PROGRAM MAIN
VAR
	bIsInitialized	: BOOL;
	//Alarms 
	fbAlarm1		: FB_TcAlarm;
	fbAlarm2		: FB_TcAlarm;
	fbAlarm3		: FB_TcAlarm;
	fbAlarm4		: FB_TcAlarm;
	fbAlarm5		: FB_TcAlarm;
	bAlarm			: BOOL;
	bClearAlarm		: BOOL;
	//Warning 
	fbWarning1 		: FB_TcAlarm;
	fbWarning2 		: FB_TcAlarm;
	fbWarning3 		: FB_TcAlarm;
	fbWarning4 		: FB_TcAlarm;
	fbWarning5 		: FB_TcAlarm;
	bWarning		: BOOL;
	bClearWarning	: BOOL;
	//Info
	fbInfo1			: FB_TcMessage;
	fbInfo2			: FB_TcMessage;
	fbInfo3			: FB_TcMessage;
	fbInfo4			: FB_TcMessage;
	fbInfo5			: FB_TcMessage;	
	bInfo			: BOOL;
	//To show alarms with arguments
	fbAlarmWithArgument1 	: FB_TcAlarm;
	fbAlarmWithArgument2 	: FB_TcAlarm;
	fErrorID1 				: LREAL := 999;
	fErrorID2 				: LREAL := 777;
	sErrorString 			: STRING := 'This is error id 777';
	bAlarmWithArg			: BOOL;
END_VAR

//Initialized the alarms, warnings and info 
IF NOT bIsInitialized THEN
	bIsInitialized := TRUE;
	fbAlarm1.CreateEx(TC_Events.MyAlarms.Alarm1, TRUE, 0);
	fbAlarm2.CreateEx(TC_Events.MyAlarms.Alarm2, TRUE, 0);
	fbAlarm3.CreateEx(TC_Events.MyAlarms.Alarm3, TRUE, 0);
	fbAlarm4.CreateEx(TC_Events.MyAlarms.Alarm4, TRUE, 0);
	fbAlarm5.CreateEx(TC_Events.MyAlarms.Alarm5, TRUE, 0);
	
	fbWarning1.CreateEx(TC_Events.InfoWarning.Warning1, TRUE, 0);
	fbWarning2.CreateEx(TC_Events.InfoWarning.Warning2, TRUE, 0);
	fbWarning3.CreateEx(TC_Events.InfoWarning.Warning3, TRUE, 0);
	fbWarning4.CreateEx(TC_Events.InfoWarning.Warning4, TRUE, 0);
	fbWarning5.CreateEx(TC_Events.InfoWarning.Warning5, TRUE, 0);
	
	fbInfo1.CreateEx(TC_Events.InfoWarning.Info1, 0);
	fbInfo2.CreateEx(TC_Events.InfoWarning.Info2, 0);
	fbInfo3.CreateEx(TC_Events.InfoWarning.Info3, 0);
	fbInfo4.CreateEx(TC_Events.InfoWarning.Info4, 0);
	fbInfo5.CreateEx(TC_Events.InfoWarning.Info5, 0);
	
	fbAlarmWithArgument1.CreateEx(TC_Events.DynamicAlarms.DynAlarm1, TRUE, 0(*fbSource*));
	fbAlarmWithArgument2.CreateEx(TC_Events.DynamicAlarms.DynAlarm2, TRUE, 0(*fbSource*));
	
END_IF 

//Trigger the alarms
IF bAlarm THEN 
	bAlarm := FALSE;
	fbAlarm1.Raise(0);
	fbAlarm2.Raise(0);
	fbAlarm3.Raise(0);
	fbAlarm4.Raise(0);
	fbAlarm5.Raise(0);
END_IF

//To raise the alarms with the arguments
IF bAlarmWithArg THEN 
	bAlarmWithArg := FALSE;
	//The arguments must be defined after Create()/CreateEx(), but before Send(), Raise()
	fbAlarmWithArgument1.ipArguments.Clear().AddLReal(fErrorID1);
	//Several arguments can be specified in concatenated form 
	fbAlarmWithArgument2.ipArguments.Clear().AddLReal(fErrorID2).AddString(sErrorString);
	//Raise the alarms
	fbAlarmWithArgument1.Raise(0);
	fbAlarmWithArgument2.Raise(0);
END_IF


//Clear all alarms 
IF bClearAlarm THEN
	bClearAlarm := FALSE;
	fbAlarm1.Clear(0, TRUE);
	fbAlarm2.Clear(0, TRUE);
	fbAlarm3.Clear(0, TRUE);
	fbAlarm4.Clear(0, TRUE);
	fbAlarm5.Clear(0, TRUE);
	
	fbAlarmWithArgument1.Clear(0, TRUE);
	fbAlarmWithArgument2.Clear(0, TRUE);
END_IF

//Raise the warnings. 
IF bWarning THEN
	bWarning := FALSE;
	fbWarning1.Raise(0);
	fbWarning2.Raise(0);
	fbWarning3.Raise(0);
	fbWarning4.Raise(0);
	fbWarning5.Raise(0);
END_IF

//Clear the warning
IF bClearWarning THEN 
	bClearWarning := FALSE;
	fbWarning1.Clear(0, TRUE);
	fbWarning2.Clear(0, TRUE);
	fbWarning3.Clear(0, TRUE);
	fbWarning4.Clear(0, TRUE);
	fbWarning5.Clear(0, TRUE);
END_IF

//Trigger the info
IF bInfo THEN 
	bInfo := FALSE;
	fbInfo1.Send(0);
	fbInfo2.Send(0);
	fbInfo3.Send(0);
	fbInfo4.Send(0);
	fbInfo5.Send(0);
END_IF

END_PROGRAM

(* stored: Version 1.1.0.1, ProductVersion 3.1.4024.4
   POU MAIN: Id {f634286c-84e3-47b0-85d8-e14e20f383c6}, SpecialFunc None *)
